Fanuc KAREL source: wdeceltol.kl

PROGRAM wdeceltol
%NOLOCKGROUP
VAR
  p : POSITION
  q : POSITION
  i : INTEGER
  r : REAL
BEGIN
  WITH $DECELTOL = 5 MOVE TO p
END wdeceltol
